TEXTLIST MoversMode_txt
  1 = 'Single'
  2 = 'Double'
  3 = 'Triple'
   = ''
END_TEXTLIST

(* stored: Version 1.1.0.1, ProductVersion 3.1.4024.11
   TextList MoversMode_txt: Id {8b475f95-fb81-41dc-ba65-88c98ad35001} *)
